{attribute 'qualified_only'}
VAR_GLOBAL
	GlobalTraceLog : FB_TraceLog;
END_VAR

(* stored: Version 1.1.0.1, ProductVersion 3.1.4024.12
   GVL Tracing: Id {9be00f29-7b5c-463b-99e8-ed1917b55319} *)
